TYPE
    TcoPlsPaletizator_Status_v_1_x_x EXTENDS TcoFeeding_Status_v_1_x_x:
    STRUCT

        {attribute addProperty Name "<#Refill required#>"}
		EntryBufferEmpty:BOOL;
		
		{attribute addProperty Name "<#Blister ready#>"}
        BlisterReady : BOOL;
		
		{attribute addProperty Name "<#Empty blisters removal required#>"}
        OutBufferFull : BOOL;
    END_STRUCT
END_TYPE

(* stored: Version 1.1.0.1
   DUT TcoPlsPaletizator_Status_v_1_x_x: Id {44e4d35e-4de6-416e-b94f-93977a6d1dd1} *)
